FUNCTION Convert_TIME_TO_TIME : Hresult
VAR_INPUT
	in : TIME;
	out : REFERENCE TO TIME;
END_VAR

out := in;

END_FUNCTION

(* stored: Version 1.1.0.1, ProductVersion 3.1.4024.12
   POU Convert_TIME_TO_TIME: Id {1b0b5518-9091-4e79-ad70-6cf7ff9751a2}, SpecialFunc None *)
